// TIA Portal V17 export
// export: Created 2025-03-05T08:02:48.265703Z, ExportSetting WithDefaults, DisplayName Totally Integrated Automation Portal, DisplayVersion V17 Update 8, DisplayName TIA Portal Openness, DisplayVersion V17 Update 8, DisplayName TIA Portal Version Control Interface, DisplayVersion V17, DisplayName SINAMICS Startdrive Advanced, DisplayVersion V17 SP2, DisplayName SINAMICS Startdrive G110M, G120, G120C, G120D, G120P, G115D, DisplayVersion V17 SP2, DisplayName SINAMICS Startdrive G130, G150, S120, S150, SINAMICS MV, S210, DisplayVersion V17 SP2, DisplayName STEP 7 Professional, DisplayVersion V17 Update 8, DisplayName SINUMERIK ONE STEP 7 Toolbox, DisplayVersion V17 Update 12, DisplayName SINUMERIK 840D sl STEP 7 Toolbox, DisplayVersion V17 Update 12, DisplayName STEP 7 Safety, DisplayVersion V17 Update 6, DisplayName WinCC Advanced, DisplayVersion V17 Update 8
DATA_BLOCK "DB2102_INFEED_MODULE"   // DB2102
{ S7_Optimized_Access := 'FALSE'; DB_Accessible_From_OPC_UA := 'FALSE' }
AUTHOR : ETXETAR
VERSION : 1.0
// stored: AutoNumber false, DBAccessibleFromOPCUA false, DBAccessibleFromWebserver true, IsOnlyStoredInLoadMemory false, IsWriteProtectedInAS false
   VAR RETAIN
      INFEED_MODULE_1_READY_I : Bool;   // INPUT 611D READY / INFEED MODULE 1 READY INPUT
      INFEED_MODULE_1_ENABLED_I : Bool;   // INPUT 611D ENABLED / INFEED MODULE 1 ENABLED INPUT
      INFEED_MODULE_1_OVERTEMPERATURE_I : Bool;   // INPUT 611D OVERTEMPERATURE / INFEED MODULE 1 OVERTEMPERATURE INPUT
      INFEED_MODULE_2_READY_I : Bool;   // INPUT 611D READY / INFEED MODULE 2 READY INPUT
      INFEED_MODULE_2_ENABLED_I : Bool;   // INPUT 611D ENABLED / INFEED MODULE 2 ENABLED INPUT
      INFEED_MODULE_2_OVERTEMPERATURE_I : Bool;   // INPUT 611D OVERTEMPERATURE / INFEED MODULE 2 OVERTEMPERATURE INPUT
      INFEED_MODULE_READY : Bool;   // POWER SUPPLY 611D READY / INFEED MODULE READY
      INFEED_MODULE_READY_ENABLE_AXES : Bool;   // POWER SUPPLY READY ENABLE AXIS / INFEED MODULE READY ENABLE AXIS
      INFEED_MODULE_1_NOT_READY_ALARM : Bool;   // POWER SUPPLY 611D NOT READY / INFEED MODULE 1 NOT READY ALARM
      INFEED_MODULE_1_OVERTEMPERATURE_ALARM : Bool;   // POWER SUPPLY 611D OVERTEMPERATURE / INFEED MODULE 1 OVERTEMPERATURE ALARM
      INFEED_MODULE_2_NOT_READY_ALARM : Bool;   // POWER SUPPLY 611D NOT READY / INFEED MODULE 2 NOT READY ALARM
      INFEED_MODULE_2_OVERTEMPERATURE_ALARM : Bool;   // POWER SUPPLY 611D OVERTEMPERATURE / INFEED MODULE 2 OVERTEMPERATURE ALARM
      NCU_HEAT_SINK_TEMPERATURE_ALARM : Bool;   // NCU TEMPERATURE FAULT / NCU HEAT SINK TEMPERATURE ALARM
      NCU_LOW_BATTERY_ALARM : Bool;   // NC BATTERY LOW / NCU LOW BATTERY ALARM
      NCU_AIR_TEMPERATURE_ALARM : Bool;   // HEAT SINK AIR FLOW FAULT / NCU AIR TEMPERATURE ALARM
      NCK_ALARM : Bool;   // NCK ALARM
      ANY_ACTIVE_ALARM : Bool;   // ANY ACTIVE ALARM
      IS_ALARMS : Bool;   // IMMEDIATE STOP ALARMS
      SEOC_ALARMS : Bool;   // STOP AT END OF CYCLE ALARMS
      INFEED_MODULE_1_NOT_READY_AUX : Bool;   // AUXILIARY NOT READY / INFEED MODULE 1 NOT READY AUXILIARY
      INFEED_MODULE_2_NOT_READY_AUX : Bool;   // AUXILIARY NOT READY / INFEED MODULE 2 NOT READY AUXILIARY
      TIMER_INFEED_MODULE_READY : TOF_TIME;   // INFEED MODULE READY TIMER
      TIMER_INFEED_MODULE_1_NOT_READY : TON_TIME;   // INFEED MODULE 1 NOT READY TIMER
      TIMER_INFEED_MODULE_2_NOT_READY : TON_TIME;   // INFEED MODULE 2 NOT READY TIMER
      TIMER_NCK_ALAR_DELAY { S7_SetPoint := 'True'} : TON_TIME;   // NCK ALARM TIMER
   END_VAR
BEGIN
   TIMER_INFEED_MODULE_READY.PT := T#1s;
   TIMER_INFEED_MODULE_1_NOT_READY.PT := T#200ms;
   TIMER_INFEED_MODULE_2_NOT_READY.PT := T#200ms;
   TIMER_NCK_ALAR_DELAY.PT := T#100ms;
END_DATA_BLOCK
